FUNCTION_BLOCK TEST_GUARDS (* Test Guard-Only Transitions *)
  (* Standard: 61499-1; Classification: Test; Description: Test Guard-Only EC Transitions *)
  (* Version 0.0, 2008-09-20, JHC, Holobloc Inc *)
  (* Compiler header: package fb.rt.test; *)
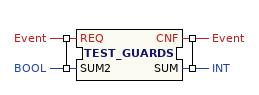
  EVENT_INPUT
    REQ WITH SUM2; (* Normal Execution Request *)
  END_EVENT
  EVENT_OUTPUT
    CNF WITH SUM; (* Execution Confirmation *)
  END_EVENT
  VAR_INPUT
    SUM2 : BOOL; (* SUM=2 if TRUE, 1 if FALSE *)
  END_VAR
  VAR_OUTPUT
    SUM : INT; (* 1 if SUM2 is FALSE, 2 if SUM2 is TRUE *)
  END_VAR
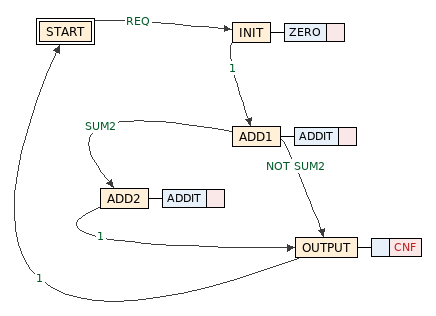
  EC_STATES
    START; (* Initial State *)
    INIT : ZERO; (* Initialize SUM to zero *)
    ADD1 : ADDIT; (* Now SUM = 1 *)
    ADD2 : ADDIT; (* Now SUM = 2 *)
    OUTPUT : -> CNF; (* Confirm result *)
  END_STATES
  EC_TRANSITIONS
    START TO INIT := REQ;
    INIT TO ADD1 := 1;
    ADD1 TO ADD2 := SUM2;
    ADD1 TO OUTPUT := NOT SUM2;
    ADD2 TO OUTPUT := 1;
    OUTPUT TO START := 1;
  END_TRANSITIONS
  ALGORITHM ZERO IN ST: (* Initialize SUM *)
SUM := 0;
  END_ALGORITHM
  ALGORITHM ADDIT IN ST: (* Add 1 to SUM *)
SUM := SUM + 1;
  END_ALGORITHM
END_FUNCTION_BLOCK
